{attribute 'linkalways'} 
{attribute 'no_explicit_call' := 'This FB is a CLASS and must be accessed using methods or properties'}
{attribute 'enable_dynamic_creation'}
FUNCTION_BLOCK FINAL SEL_ULINT EXTENDS Node
VAR
	g : _BOOL(FALSE);
	in1 : _ULINT(0);
	in2 : _ULINT(0);
	out : _ULINT(0);
END_VAR

METHOD PUBLIC Clone : I_Node
VAR
	pNode : POINTER TO SEL_ULINT;
END_VAR
pNode := __NEW(SEL_ULINT);
Clone := pNode^;
END_METHOD

METHOD FB_init : BOOL
VAR_INPUT
	bInitRetains : BOOL; // if TRUE, the retain variables are initialized (warm start / cold start)
	bInCopyCode : BOOL;  // if TRUE, the instance afterwards gets moved into the copy code (online change)
END_VAR
AddInput('g',THIS^.g);
AddInput('in1',THIS^.in1);
AddInput('in2',THIS^.in2);
AddOutput('out', THIS^.out);
END_METHOD

METHOD PROTECTED OnExecute
VAR
END_VAR
IF g.value THEN
	out.value := in2.value;
ELSE
	out.value := in1.value;
END_IF
END_METHOD

END_FUNCTION_BLOCK

(* stored: Version 1.1.0.1, ProductVersion 3.1.4024.15
   POU SEL_ULINT: Id {963218fa-a3db-4315-9740-43f5156ef583}, SpecialFunc None
   Folder Constructor: Id {67deb5e6-f833-4f70-b8ba-2904d6071c14}
   Method Clone: Id {57105159-0e6d-4405-af98-fc0d1fa6b54f}
   Method FB_init: Id {eea64183-b190-4cc2-ac37-c4ee364b07b9}
   Method OnExecute: Id {2e9f04a0-703d-4b47-b721-b46b09c3d502} *)
